// TIA Portal project "water_tank_timer" (V19)

(* hardware
DEVICE "S7-1200 station_1"  S7-1200 Station
   slot 0: "Rack_0"  S7-1200 Rack  Rack  V1.0
   slot 1: "PLC_1"  CPU 1212C DC/DC/Rly  6ES7 212-1HE40-0XB0  V4.5
*)

// ===== PLC "PLC_1"  CPU 1212C DC/DC/Rly =====

VAR_GLOBAL   // PLC tag table "Default tag table"
   "Fill" AT %I0.0 : Bool;
   "Discharge" AT %I0.1 : Bool;
   "Start" AT %I0.2 : Bool;
   "Fill valve" AT %Q0.0 : Bool;
   "Discharge valve" AT %Q0.2 : Bool;
   "Fill flag" AT %M0.0 : Bool;
   "Discharge flag" AT %M0.1 : Bool;
   "Filling Light" AT %Q0.1 : Bool;
   "Discharging Light" AT %Q0.3 : Bool;
   "Fill Timer" AT %MD0 : Time;
   "Discharge finish" AT %M0.3 : Bool;
END_VAR

// folder: System blocks/Program resources

DATA_BLOCK "IEC_Timer_0_DB"   // DB1
{ S7_Optimized_Access := 'TRUE' }
AUTHOR : Simatic
FAMILY : IEC
NAME : IEC_TMR
VERSION : 1.0
// stored: InstanceOfName IEC_TIMER
"IEC_TIMER"
BEGIN
END_DATA_BLOCK

DATA_BLOCK "IEC_Timer_0_DB_1"   // DB2
{ S7_Optimized_Access := 'TRUE' }
AUTHOR : Simatic
FAMILY : IEC
NAME : IEC_TMR
VERSION : 1.0
// stored: InstanceOfName IEC_TIMER
"IEC_TIMER"
BEGIN
END_DATA_BLOCK

// folder: (top level)

ORGANIZATION_BLOCK "Main"   // OB1, LAD, ProgramCycle
TITLE = "Main Program Sweep (Cycle)"
{ S7_Optimized_Access := 'TRUE' }
VERSION : 0.1
   VAR_INPUT
      Initial_Call : Bool;   // Initial call of this OB
      Remanence : Bool;   // =True, if remanent data are available
   END_VAR
BEGIN

REGION Network 1
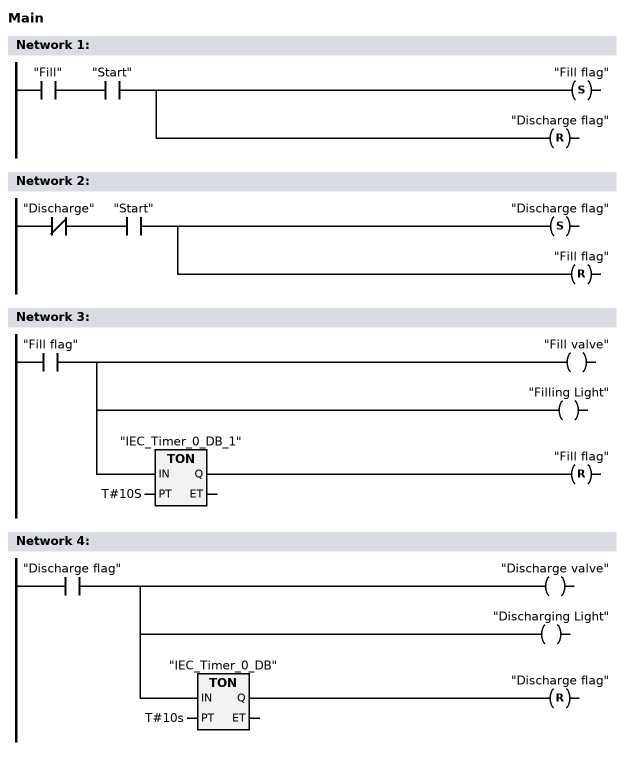
   RUNG wire#powerrail
      Contact( "Fill" )
      Contact( "Start" )
      wire#w1
      S_Coil( "Fill flag" )
   END_RUNG
   RUNG wire#w1
      R_Coil( "Discharge flag" )
   END_RUNG
   // the same network as SCL:
   IF "Fill" AND "Start" THEN
       "Fill flag" := TRUE;
       "Discharge flag" := FALSE;
   END_IF;
END_REGION

REGION Network 2
   RUNG wire#powerrail
      I_Contact( "Discharge" )
      Contact( "Start" )
      wire#w1
      S_Coil( "Discharge flag" )
   END_RUNG
   RUNG wire#w1
      R_Coil( "Fill flag" )
   END_RUNG
   // the same network as SCL:
   IF NOT "Discharge" AND "Start" THEN
       "Discharge flag" := TRUE;
       "Fill flag" := FALSE;
   END_IF;
END_REGION

REGION Network 3
   "Fill valve" := "Fill flag";
   "Filling Light" := "Fill flag";
   "IEC_Timer_0_DB_1".TON(IN := "Fill flag", PT := T#10S);
   IF "IEC_Timer_0_DB_1".Q THEN "Fill flag" := FALSE; END_IF;
END_REGION

REGION Network 4
   "Discharge valve" := "Discharge flag";
   "Discharging Light" := "Discharge flag";
   "IEC_Timer_0_DB".TON(IN := "Discharge flag", PT := T#10s);
   IF "IEC_Timer_0_DB".Q THEN "Discharge flag" := FALSE; END_IF;
END_REGION
END_ORGANIZATION_BLOCK